Staubli VAL3: new.pgx

public program new(trsf& tPar[])
  local num nSize
  local tool tGun
begin
  // only fifo polit
  call getSize(nSize)
  // TRSF
  $dins(saveTool:gun,nSize)
  tGun.trsf=tPar
  call setTool(tGun,nSize)
  // NAME
  $dins(saveTool:name,nSize)
  call setName("",nSize)
  // ACTION
  $dins(saveTool:sActionON,nSize)
  $dins(saveTool:sActionOFF,nSize)
end
